TYPE "PPrf_A02_S1_PartsCutting"
VERSION : 0.1
// Block: PPrf_A02_S1_PartsCutting
   STRUCT
      Rollformer : PPrf_Rollformer;
   END_STRUCT;

END_TYPE
